{attribute addProperty BoxType "EP8309-0022-0021"}
{attribute addProperty Id "Reset_ErrorAT %Q*BOOL81"}
{attribute addProperty CRC "579923262"}
{attribute addProperty SizeInBites "8"}
{attribute addProperty SizeInBytes "1"}
TYPE TACHO_Output_Channel_2290ED3E :
STRUCT
	{attribute addProperty Name "Reset_Error"}
	Reset_Error AT %Q* : BOOL;
END_STRUCT
END_TYPE

(* stored: Version 1.2.0.0, ProductVersion 3.1.4024.9
   DUT TACHO_Output_Channel_2290ED3E: Id {5d26322e-e52f-4fcc-a298-da9eecb3eff6} *)
